// TwinCAT 3 PLC project TcoKukaRobotics
// Title: TcoKukaRobotics
// Company: Vortex.Library
// Author: TcOpenGroup
// ProjectVersion: 0.6.0.913
// ProgramVersion: 3.1.4024.12
// libraries:
//   Tc2_MC2, * (Beckhoff Automation GmbH)
//   Tc2_MC2_Drive, * (Beckhoff Automation GmbH)
//   Tc2_Standard, * (Beckhoff Automation GmbH)
//   Tc2_System, * (Beckhoff Automation GmbH)
//   Tc3_Module, * (Beckhoff Automation GmbH)
//   TcoAbstractions, 0.6.0.913 (Vortex.Library)
//   TcoCore, 0.6.0.913 (Vortex.Library)
//   TcoIo, 0.6.0.913 (Vortex.Library)
//   TcoUtilities, 0.6.0.913 (Vortex.Library)
// project tree:
//   DUTs/ TcoKukaRobotics_Config_v_5_x_x.TcDUT, TcoKukaRobotics_Control_v_5_x_x.TcDUT, TcoKukaRobotics_State_v_5_x_x.TcDUT, TcoKukaRobotics_Status_v_5_x_x.TcDUT
//   / PlcTask.TcTTO
//   POUs/ MAIN.TcPOU
//   POUs/Prototypes/KRC4/IO/ TcoKrc4_Inputs_v_5_x_x.TcDUT, TcoKrc4_IO_v_5_x_x.TcDUT, TcoKrc4_Outputs_v_5_x_x.TcDUT
//   POUs/Prototypes/KRC4/ TcoKrc4_v_5_x_x.TcPOU
//   POUs/Prototypes/RoboticsTasks/Starts/ StartAtMainTask.TcPOU, StartMotorsAndProgramTask.TcPOU, StartMotorsProgramAndMovementsTask.TcPOU, StartMotorsTask.TcPOU, StartMovementsTask.TcPOU, StartProgramTask.TcPOU
//   POUs/Prototypes/RoboticsTasks/Stops/ StopMotorsTask.TcPOU, StopMovementsAndProgramTask.TcPOU, StopMovementsTask.TcPOU, StopProgramTask.TcPOU
//   POUs/Prototypes/RoboticsTasks/ TcoKukaRoboticsTask.TcPOU
// real-time tasks:
//   TASK PlcTask: cycle T#10ms, priority 20, ADS port 350
//   TASK PlcTask1: cycle T#10ms, priority 1, ADS port 351
//   TASK PN: cycle T#8ms, priority 2, ADS port 301
// I/O:
//   DEVICE Device 4 (EtherCAT) (disabled), AmsNetId 172.20.10.104.5.1
//     Term 1 (EK1100) [EK1100 EtherCAT Coupler (2A E-Bus)]
//       Term 2 (EL1008) [EL1008 8Ch. Dig. Input 24V, 3ms]
//       Term 3 (EL2008) [EL2008 8Ch. Dig. Output 24V, 0.5A]
//       Term 4 (EL3052) [EL3052 2Ch. Ana. Input 4-20mA]
//       Term 5 (EL9576) [EL9576 Brake chopper terminal]
//       Term 6 (EL7211-0010) [EL7211-0010 1Ch. MDP742 Servo motor output stage with OCT (50V, 4.5A RMS)]
//       Term 14 (EL7047) [EL7047 1Ch. Stepper motor output stage (50V, 5A)]
//       Term 8 (EL9011) [EL9011 End Terminal]
//   DEVICE Device 1 (EtherCAT) (disabled), AmsNetId 192.168.4.1.2.1
//     Drive 7 (IndraDrive MPB20) [IndraDrive MPB20]
//   DEVICE Device 2 (EtherCAT) (disabled), AmsNetId 192.168.4.1.3.1
//     Term 1 (EK1200) [EK1200-5000 EtherCAT Power supply (2A E-Bus)]
//       Term 10 (EK1122) [EK1122 2 port EtherCAT junction]
//       Term 13 (EL6631) [EL6631 PROFINET IO Controller]
//       Term 12 (EL1809) [EL1809 16Ch. Dig. Input 24V, 3ms]
//       Term 13 (EL2809) [EL2809 16Ch. Dig. Output 24V, 0.5A]
//       Term 15 (EL4004) [EL4004 4Ch. Ana. Output 0-10V, 12bit]
//       Term 16 (EL7342) [EL7342 2Ch. DC motor output stage (50V, 3.5A)]
//       Term 17 (EL4004) [EL4004 4Ch. Ana. Output 0-10V, 12bit]
//       Term 18 (EL6001) [EL6001 Interface (RS232)]
//       Term 10 (EL9011) [EL9011 End Terminal]
//   DEVICE Device 3 (EL6631) (disabled), AmsNetId 192.168.4.1.4.1
//     krc4 [KUKA Roboter GmbH PROFINET IO 0x300]
//       modules: Term 4 (DAP Module), Term 5 (64 safe digital in- and outputs), Term 6 (512 digital in- and outputs)
// variable links:
//   TcoKukaRoboticsTests/TcoKukaRoboticsTests Instance <-> Device 3 (EL6631)/krc4
//     PlcTask1 Inputs/GVL.Robot1.In.Inputs[{0..63}] <-> API/Term 6 (512 digital in- and outputs)/Subterm 10 (512 digital in- and outputs)/Inputs/8 digital inputs[{0..63}]  (64 links)
//     PlcTask1 Inputs/GVL.Robot1.PnIoBoxDiag <-> Inputs/PnIoBoxDiag
//     PlcTask1 Inputs/GVL.Robot1.PnIoBoxState <-> Inputs/PnIoBoxState
//     PlcTask1 Outputs/GVL.Robot1.Out.Outputs[{0..63}] <-> API/Term 6 (512 digital in- and outputs)/Subterm 10 (512 digital in- and outputs)/Outputs/8 digital outputs[{0..63}]  (64 links)

CONFIGURATION TcoKukaRobotics
    RESOURCE PLC ON TwinCAT3
        TASK PlcTask(INTERVAL := T#10ms, PRIORITY := 20);
        PROGRAM MAIN WITH PlcTask : MAIN;
    END_RESOURCE
END_CONFIGURATION

// ---- DUTs/TcoKukaRobotics_Config_v_5_x_x.TcDUT
TYPE TcoKukaRobotics_Config_v_5_x_x :
STRUCT
    InfoTime : TIME := T#2S;
    ErrorTime : TIME := T#0S;
END_STRUCT
END_TYPE

// ---- DUTs/TcoKukaRobotics_Control_v_5_x_x.TcDUT
TYPE TcoKukaRobotics_Control_v_5_x_x :
STRUCT
    {attribute addProperty Name "<#Program Start [EXT_START]#>"}
    ExternalStart : BOOL;
    {attribute addProperty Name "<#Move Enable [MOVE_ENABLE]#>"}
    MoveEnable : BOOL;
    {attribute addProperty Name "<#Error Confirmation [CONF_MESS]#>"}
    ErrorConfirmation : BOOL;
    {attribute addProperty Name "<#Drives Off [DRIVES_OFF]#>"}
    DrivesOff : BOOL;
    {attribute addProperty Name "<#Drives On [DRIVES_ON]#>"}
    DrivesOn : BOOL;
    {attribute addProperty Name "<#Activate Interface [I_O_ACT]#>"}
    ActivateInterface : BOOL;
    {attribute addProperty Name "<#Start At Main [START_AT_MAIN]#>"}
    StartAtMain : BOOL;
    {attribute addProperty Name "<#Master mode#>"}
    MasterMode : BYTE;
    {attribute addProperty Name "<#Tool 1 retract#>"}
    Tool_1_Retract : BOOL;
    {attribute addProperty Name "<#Tool 1 extend#>"}
    Tool_1_Extend : BOOL;
    {attribute addProperty Name "<#Tool 2 retract#>"}
    Tool_2_Retract : BOOL;
    {attribute addProperty Name "<#Tool 2 extend#>"}
    Tool_2_Extend : BOOL;
    {attribute addProperty Name "<#Tool 3 retract#>"}
    Tool_3_Retract : BOOL;
    {attribute addProperty Name "<#Tool 3 extend#>"}
    Tool_3_Extend : BOOL;
    {attribute addProperty Name "<#Tool 4 retract#>"}
    Tool_4_Retract : BOOL;
    {attribute addProperty Name "<#Tool 4 extend#>"}
    Tool_4_Extend : BOOL;
    {attribute addProperty Name "<#Zones#>"}
    Zone : BYTE;
    {attribute addProperty Name "<#In position#>"}
    InPosition : BYTE;
    {attribute addProperty Name "<#Action number#>"}
    ActionNo : BYTE;
    {attribute addProperty Name "<#Global robot speed#>"}
    GlobalSpeed : BYTE;
    {attribute addProperty Name "<#Tool number#>"}
    ToolNo : BYTE;
    {attribute addProperty Name "<#Workobject number#>"}
    WorkobjectNo : BYTE;
    {attribute addProperty Name "<#Point number#>"}
    PointNo : BYTE;
    {attribute addProperty Name "<#User specific speed 1#>"}
    UserSpecSpeed1 : REAL;
    {attribute addProperty Name "<#User specific speed 2#>"}
    UserSpecSpeed2 : REAL;
    {attribute  addProperty Name "<#Coordinates#>"}
    Coordinates : TcoAbstractions.TcoRoboticsCoordinates;
END_STRUCT
END_TYPE

// ---- DUTs/TcoKukaRobotics_State_v_5_x_x.TcDUT
TYPE TcoKukaRobotics_State_v_5_x_x :
STRUCT
    {attribute addProperty Name "<#ControlReady [RC_RDY1]#>"}
    RcReady : BOOL;
    {attribute addProperty Name "<#AlarmStopActive [ALARM_STOP]#>"}
    AlarmStopActive : BOOL;
    {attribute addProperty Name "<#UserSafetySwitchClosed [USER_SAF]#>"}
    UserSafetySwitchClosed : BOOL;
    {attribute addProperty Name "<#DrivesReady [PERI_RDY]#>"}
    DrivesReady : BOOL;
    {attribute addProperty Name "<#RobotCalibrated [ROB_CAL]#>"}
    RobotCalibrated : BOOL;
    {attribute addProperty Name "<#InterfaceActivated [I_O_ACTCONF]#>"}
    InterfaceActivated : BOOL;
    {attribute addProperty Name "<#ErrorCollection [STOPMESS]#>"}
    StopMess : BOOL;
    {attribute addProperty Name "<#RobotStopped [ROB_STOPPED]#>"}
    RobotStopped : BOOL;
    {attribute addProperty Name "<#InHome [IN_HOME]#>"}
    InHome : BOOL;
    {attribute addProperty Name "<#Manual [T1]#>"}
    Manual : BOOL;
    {attribute addProperty Name "<#Automatic [AUT]#>"}
    Automatic : BOOL;
    {attribute addProperty Name "<#ExternalAutomatic [EXT]#>"}
    ExternalAutomatic : BOOL;
    {attribute addProperty Name "<#ProcesActive [PRO_ACT]#>"}
    ProActive : BOOL;
    {attribute addProperty Name "<#ProgramMoveActive [PROGRAM MOVEMENT ACTIVE]#>"}
    ProgramMoveActive : BOOL;
    {attribute addProperty Name "<#Event ID#>"}
    EventId : UDINT;
    {attribute addProperty Name "<#PpMoved#>"}
    PpMoved : BOOL;
    {attribute addProperty Name "<#StartAtMain#>"}
    StartAtMain : BOOL;
    {attribute addProperty Name "<#Error#>"}
    Error : BOOL;
    {attribute addProperty Name "<#In area 1#>"}
    InArea_1 : BOOL;
    {attribute addProperty Name "<#In area 2#>"}
    InArea_2 : BOOL;
    {attribute addProperty Name "<#In area 3#>"}
    InArea_3 : BOOL;
    {attribute addProperty Name "<#In area 4#>"}
    InArea_4 : BOOL;
    {attribute addProperty Name "<#In position 1#>"}
    InPosition_1 : BOOL;
    {attribute addProperty Name "<#In position 2#>"}
    InPosition_2 : BOOL;
    {attribute addProperty Name "<#In position 3#>"}
    InPosition_3 : BOOL;
    {attribute addProperty Name "<#In position 4#>"}
    InPosition_4 : BOOL;
    {attribute addProperty Name "<#Zones#>"}
    Zone : BYTE;
    {attribute addProperty Name "<#In position#>"}
    InPosition : BYTE;
    {attribute addProperty Name "<#Tool 1 retract#>"}
    Tool_1_Retract : BOOL;
    {attribute addProperty Name "<#Tool 1 extend#>"}
    Tool_1_Extend : BOOL;
    {attribute addProperty Name "<#Tool 2 retract#>"}
    Tool_2_Retract : BOOL;
    {attribute addProperty Name "<#Tool 2 extend#>"}
    Tool_2_Extend : BOOL;
    {attribute addProperty Name "<#Tool 3 retract#>"}
    Tool_3_Retract : BOOL;
    {attribute addProperty Name "<#Tool 3 extend#>"}
    Tool_3_Extend : BOOL;
    {attribute addProperty Name "<#Tool 4 retract#>"}
    Tool_4_Retract : BOOL;
    {attribute addProperty Name "<#Tool 4 extend#>"}
    Tool_4_Extend : BOOL;
    {attribute addProperty Name "<#Action number#>"}
    ActionNo : BYTE;
    {attribute addProperty Name "<#Global speed#>"}
    GlobalSpeed : BYTE;
    {attribute addProperty Name "<#Tool number#>"}
    ToolNo : BYTE;
    {attribute addProperty Name "<#Workobject number#>"}
    WorkobjectNo : BYTE;
    {attribute addProperty Name "<#PointNumber#>"}
    PointNo : BYTE;
    {attribute addProperty Name "<#User specific speed 1#>"}
    UserSpecSpeed1 : DINT;
    {attribute addProperty Name "<#User specific speed 2#>"}
    UserSpecSpeed2 : DINT;
    {attribute  addProperty Name "<#Coordinates#>"}
    Coordinates : TcoAbstractions.TcoRoboticsCoordinates;
END_STRUCT
END_TYPE

// ---- DUTs/TcoKukaRobotics_Status_v_5_x_x.TcDUT
TYPE TcoKukaRobotics_Status_v_5_x_x :
STRUCT
    ActionDescription : STRING(100);
    State : TcoKukaRobotics_State_v_5_x_x;
END_STRUCT
END_TYPE

// ---- POUs/Prototypes/KRC4/IO/TcoKrc4_Inputs_v_5_x_x.TcDUT
TYPE TcoKrc4_Inputs_v_5_x_x :
STRUCT
    Inputs AT %I* : ARRAY[0..63] OF BYTE;
END_STRUCT
END_TYPE

// ---- POUs/Prototypes/KRC4/IO/TcoKrc4_IO_v_5_x_x.TcDUT
TYPE TcoKrc4_IO_v_5_x_x :
STRUCT
    PnIoBoxState AT %I* : UINT;
    PnIoBoxDiag AT %I* : UINT;
    PnIoBoxCtrl AT %Q* : UINT;
    {attribute addProperty Name "<#IN#>"}
    In : TcoKrc4_Inputs_v_5_x_x;
    {attribute addProperty Name "<#OUT#>"}
    Out : TcoKrc4_Outputs_v_5_x_x;
END_STRUCT
END_TYPE

// ---- POUs/Prototypes/KRC4/IO/TcoKrc4_Outputs_v_5_x_x.TcDUT
TYPE TcoKrc4_Outputs_v_5_x_x :
STRUCT
    Outputs AT %Q* : ARRAY[0..63] OF BYTE;
END_STRUCT
END_TYPE

// ---- POUs/MAIN.TcPOU
PROGRAM MAIN
VAR
END_VAR

END_PROGRAM

// ---- POUs/Prototypes/KRC4/TcoKrc4_v_5_x_x.TcPOU
FUNCTION_BLOCK TcoKrc4_v_5_x_x EXTENDS TcoIo.TcoPnIoComponent IMPLEMENTS TcoAbstractions.ITcoRobotics
VAR_INPUT
    inEnable : BOOL;
END_VAR
VAR_OUTPUT
END_VAR
VAR_IN_OUT
    inoData : TcoKrc4_IO_v_5_x_x;
END_VAR
VAR
    {attribute addProperty Name "<#Status#>"}
    {attribute clr [ReadOnly()]}
    _status : TcoKukaRobotics_Status_v_5_x_x;
    {attribute addProperty Name "<#Control#>"}
    _control : TcoKukaRobotics_Control_v_5_x_x;
    {attribute addProperty Name "<#Config#>"}
    _config : TcoKukaRobotics_Config_v_5_x_x;
    {attribute addProperty Name "<#PN Error#>"}
    {attribute clr [ReadOnly()]}
    _pnError : BOOL;
    _someTaskIsActive : BOOL;
    _stopTasksAreActive : BOOL;
END_VAR
VAR
    {attribute addProperty Name "<#Start at Main#>"}
    _startAtMainTask : StartAtMainTask(THIS^);
    {attribute addProperty Name "<#Start motors and program#>"}
    _startMotorsAndProgramTask : StartMotorsAndProgramTask(THIS^);
    {attribute addProperty Name "<#Start program#>"}
    _startProgramTask : StartProgramTask(THIS^);
    {attribute addProperty Name "<#Start motors#>"}
    _startMotorsTask : StartMotorsTask(THIS^);
    {attribute addProperty Name "<#Start movements#>"}
    _startMovementsTask : StartMovementsTask(THIS^);
    {attribute addProperty Name "<#Start motors program and movements#>"}
    _startMotorsProgramAndMovementsTask : StartMotorsProgramAndMovementsTask(THIS^);
    {attribute addProperty Name "<#Stop movements#>"}
    _stopMovementsTask : StopMovementsTask(THIS^);
    {attribute addProperty Name "<#Stop movenents and program#>"}
    _stopMovementsAndProgramTask : StopMovementsAndProgramTask(THIS^);
    {attribute addProperty Name "<#Stop program#>"}
    _stopProgramTask : StopProgramTask(THIS^);
    {attribute addProperty Name "<#Stop motors#>"}
    _stopMotorsTask : StopMotorsTask(THIS^);
    {attribute addProperty Name "<#Restore#>"}
    _restoreTask : TcoCore.TcoTask(THIS^);
END_VAR
VAR
    {attribute 'hide'}
    _sb : TcoCore.StringBuilder;
END_VAR

IF NOT __ISVALIDREF(inoData) THEN
    Messenger.Post('Invalid reference', TcoCore.eMessageCategory.ProgrammingError);
    RETURN;
END_IF

SUPER^(inPnIoBoxState := THIS^.inoData.PnIoBoxState, inPnIoBoxDiag := THIS^.inoData.PnIoBoxDiag);
_pnError := not _profinetReady;
UpdateStatus();
_stopTasksAreActive := _stopMovementsTask.Busy AND _stopMovementsAndProgramTask.Busy AND _stopProgramTask.Busy AND _stopMotorsTask.Busy;
_startAtMainTask.Enabled := NOT _stopTasksAreActive;
_startAtMainTask(inoConfig := _config, inoControl := _control, inoStatus := _status);
_startProgramTask.Enabled := NOT _stopTasksAreActive;
_startProgramTask(inoConfig := _config, inoControl := _control, inoStatus := _status);
_startMotorsTask.Enabled := NOT _stopTasksAreActive AND NOT _startMotorsProgramAndMovementsTask.Busy AND NOT _startMotorsAndProgramTask.Busy;
_startMotorsTask(inoConfig := _config, inoControl := _control, inoStatus := _status);
_startMotorsAndProgramTask.Enabled := NOT _stopTasksAreActive AND NOT _startProgramTask.Busy AND NOT _startMotorsTask.Busy;
_startMotorsAndProgramTask(inoConfig := _config, inoControl := _control, inoStatus := _status);
_startMovementsTask.Enabled := NOT _startMotorsProgramAndMovementsTask.Busy AND NOT _stopMotorsTask.Busy;
_startMovementsTask(inoConfig := _config, inoControl := _control, inoStatus := _status);
_startMotorsProgramAndMovementsTask.Enabled := NOT _startMovementsTask.Busy AND NOT _stopMotorsTask.Busy;

_startMotorsProgramAndMovementsTask(refStartMotorsAndProgramTask := _startMotorsAndProgramTask,
    inoConfig := _config,
    inoControl := _control,
    inoStatus := _status);

_stopMovementsTask.Enabled := TRUE;
_stopMovementsTask(inoConfig := _config, inoControl := _control, inoStatus := _status);
_stopMotorsTask.Enabled := TRUE;
_stopMotorsTask(inoConfig := _config, inoControl := _control, inoStatus := _status);
_stopProgramTask.Enabled := TRUE;
_stopProgramTask(inoConfig := _config, inoControl := _control, inoStatus := _status);
_stopMovementsAndProgramTask.Enabled := NOT _stopProgramTask.Busy AND NOT _stopProgramTask.Busy;
_stopMovementsAndProgramTask(inoConfig := _config, inoControl := _control, inoStatus := _status);
//*************RESTORE********************
_restoreTask.Enabled := TRUE;

IF _restoreTask.Execute() THEN
    Restore();
    _restoreTask.DoneWhen(TRUE);
END_IF

//****************************************
_someTaskIsActive := _startAtMainTask.Busy OR
    _startMotorsAndProgramTask.Busy OR
    _startMovementsTask.Busy OR
    _startMovementsTask.Busy OR
    _stopMovementsTask.Busy OR
    _stopMovementsAndProgramTask.Busy OR
    _stopProgramTask.Busy;

//do not publish diagnostic message when component is not used
IF _someTaskIsActive THEN
    IF (NOT _status.State.AlarmStopActive) THEN
        Messenger.Error('<#Emergency stop active#>');
    END_IF;

    IF (NOT _status.State.UserSafetySwitchClosed) THEN
        Messenger.Warning('<#Safety Error #>');
    END_IF;
END_IF;

IF (_status.State.Error) THEN
    Messenger.Error(_sb.Clear()
            .Append('<#Robot reported an error: #>')
            .Append(UDINT_TO_STRING(_status.State.EventId))
            .Append(' |[[0]AdvancedDiagnosticMessage]|')
            .Append('.')
            .Append('For details see the service mode')
            .ToString());
END_IF;

UpdateControl();

(*~
    <docu>
        <summary>
            Gets the configuration of the IRC 5.
        </summary>
    </docu>
~*)
PROPERTY Config : REFERENCE TO TcoKukaRobotics_Config_v_5_x_x
GET
Config REF= _config;
END_GET
END_PROPERTY

PROPERTY PUBLIC Control : REFERENCE TO TcoKukaRobotics_Control_v_5_x_x
GET
Control REF= _control;
END_GET
END_PROPERTY

METHOD FB_init : BOOL
VAR_INPUT
    bInitRetains : BOOL; // if TRUE, the retain variables are initialized (warm start / cold start)
    bInCopyCode : BOOL; // if TRUE, the instance afterwards gets moved into the copy code (online change)
    ParentObject : ITcoObject;
END_VAR
END_METHOD

(*~
    <docu>
        <summary>
            Restores this instance to the Ready state. Can be called explicitly or from within one of the restore mechanisms.
        </summary>
    </docu>
~*)
METHOD Restore : ITcoRestorable
RestoreTasks();
_control.GlobalSpeed := 0;
_control.ActivateInterface := FALSE;
_control.ErrorConfirmation := FALSE;
_control.ExternalStart := FALSE;
_control.MasterMode := 0;
//todo to restore control signals
_control.ToolNo := 0;
_control.WorkobjectNo := 0;
_control.PointNo := 0;
_control.UserSpecSpeed1 := 0;
_control.UserSpecSpeed2 := 0;
_control.Coordinates.X := 0;
_control.Coordinates.Y := 0;
_control.Coordinates.Z := 0;
_control.Coordinates.Rx := 0;
_control.Coordinates.Ry := 0;
_control.Coordinates.Rz := 0;
END_METHOD

METHOD INTERNAL RestoreTasks
//_resetTask.Restore();
_startAtMainTask.Restore();
_startMovementsTask.Restore();
_startProgramTask.Restore();
_startMotorsTask.Restore();
_stopMotorsTask.Restore();
_startMotorsProgramAndMovementsTask.Restore();
_stopMovementsTask.Restore();
_startMotorsAndProgramTask.Restore();
_stopMovementsAndProgramTask.Restore();
_stopProgramTask.Restore();
END_METHOD

(*~
    <docu>
        <summary>
            Custom service (manual, maintenance) logic.
            This method must be implemented in derived class.
        </summary>
    </docu>
~*)
METHOD PROTECTED ServiceMode
END_METHOD

METHOD PUBLIC StartAtMain : TcoCore.ITcoTaskStatus
VAR_INPUT
END_VAR
StartAtMain := _startAtMainTask.Invoke();
END_METHOD

PROPERTY StartAtMainTask : TcoCore.ITcoTaskStatus
GET
StartAtMainTask := _startAtMainTask;
END_GET
END_PROPERTY

METHOD PUBLIC StartMotors : TcoCore.ITcoTaskStatus
StartMotors := _startMotorsTask.Invoke();
END_METHOD

METHOD StartMotorsAndProgram : TcoCore.ITcoTaskStatus
VAR_INPUT
END_VAR
StartMotorsAndProgram := THIS^._startMotorsAndProgramTask.Invoke();
END_METHOD

PROPERTY StartMotorsAndProgramTask : TcoCore.ITcoTaskStatus
GET
StartMotorsAndProgramTask := _startMotorsAndProgramTask;
END_GET
END_PROPERTY

METHOD PUBLIC StartMotorsProgramAndMovements : TcoCore.ITcoTaskStatus
VAR_INPUT
    inData : TcoRoboticsMovementsParams;
END_VAR
StartMotorsProgramAndMovements := _startMotorsProgramAndMovementsTask.InvokeWithParams(inData);
END_METHOD

PROPERTY StartMotorsProgramAndMovementsTask : TcoCore.ITcoTaskStatus
GET
StartMotorsProgramAndMovementsTask := _startMotorsProgramAndMovementsTask;
END_GET
END_PROPERTY

PROPERTY StartMotorsTask : TcoCore.ITcoTaskStatus
GET
StartMotorsTask := _startMotorsTask;
END_GET
END_PROPERTY

METHOD PUBLIC StartMovements : TcoCore.ITcoTaskStatus
VAR_INPUT
    inData : TcoRoboticsMovementsParams;
END_VAR
StartMovements := _startMovementsTask.InvokeWithParams(inData);
END_METHOD

PROPERTY StartMovementsTask : TcoCore.ITcoTaskStatus
GET
StartMovementsTask := _startMovementsTask;
END_GET
END_PROPERTY

METHOD PUBLIC StartProgram : TcoCore.ITcoTaskStatus
StartProgram := _startProgramTask.Invoke();
END_METHOD

PROPERTY StartProgramTask : TcoCore.ITcoTaskStatus
GET
StartProgramTask := _startProgramTask;
END_GET
END_PROPERTY

(*~
    <docu>
        <summary>
            Gets the status of the IRC5.
        </summary>
    </docu>
~*)
PROPERTY Status : REFERENCE TO TcoKukaRobotics_Status_v_5_x_x
GET
Status REF= _status;
END_GET
END_PROPERTY

METHOD PUBLIC StopMotors : TcoCore.ITcoTaskStatus
StopMotors := _stopMotorsTask.Invoke();
END_METHOD

PROPERTY StopMotorsTask : TcoCore.ITcoTaskStatus
GET
StopMotorsTask := _stopMotorsTask;
END_GET
END_PROPERTY

METHOD PUBLIC StopMovements : TcoCore.ITcoTaskStatus
VAR_INPUT
    inStopType : eTcoRoboticsStopType;
END_VAR
StopMovements := _stopMovementsTask.InvokeWithParams(inStopType);
END_METHOD

METHOD PUBLIC StopMovementsAndProgram : TcoCore.ITcoTaskStatus
VAR_INPUT
    inStopType : eTcoRoboticsStopType;
END_VAR
StopMovementsAndProgram := _stopMovementsAndProgramTask.InvokeWithParams(inStopType);
END_METHOD

PROPERTY StopMovementsAndProgramTask : TcoCore.ITcoTaskStatus
GET
StopMovementsAndProgramTask := _stopMovementsAndProgramTask;
END_GET
END_PROPERTY

PROPERTY StopMovementsTask : TcoCore.ITcoTaskStatus
GET
StopMovementsTask := _stopMovementsTask;
END_GET
END_PROPERTY

METHOD PUBLIC StopProgram : TcoCore.ITcoTaskStatus
StopProgram := _stopProgramTask.Invoke();
END_METHOD

PROPERTY StopProgramTask : TcoCore.ITcoTaskStatus
GET
StopProgramTask := _stopProgramTask;
END_GET
END_PROPERTY

METHOD INTERNAL UpdateControl
VAR_INPUT
END_VAR
VAR
    index : INT;
END_VAR
//SYSTEM OUTPUTS
index := 0;
inoData.Out.Outputs[index].0 := _control.ExternalStart;
inoData.Out.Outputs[index].1 := _control.MoveEnable;
inoData.Out.Outputs[index].2 := _control.ErrorConfirmation;
inoData.Out.Outputs[index].3 := _control.DrivesOff;
inoData.Out.Outputs[index].4 := _control.DrivesOn;
inoData.Out.Outputs[index].5 := _control.ActivateInterface;
inoData.Out.Outputs[index].6 := _control.StartAtMain;
//index:=1;
//inoData.Out.Outputs[index].0 	:= 		_control.StartProgram;
//inoData.Out.Outputs[index].1 	:= 		_control.StartAtMain;
//inoData.Out.Outputs[index].2 	:= 		_control.StopProgram;
//inoData.Out.Outputs[index].3 	:= 		_control.QuickStop;
//inoData.Out.Outputs[index].4 	:= 		_control.SoftStop;
//inoData.Out.Outputs[index].5 	:= 		_control.StopCycle;
//inoData.Out.Outputs[index].6 	:= 		_control.StopInstruction;
//inoData.Out.Outputs[index].7 	:= 		_control.LimitSpeed;
//Tool signals
index := 2;
inoData.Out.Outputs[index].0 := _control.Tool_1_Retract;
inoData.Out.Outputs[index].1 := _control.Tool_1_Extend;
inoData.Out.Outputs[index].2 := _control.Tool_2_Retract;
inoData.Out.Outputs[index].3 := _control.Tool_2_Extend;
inoData.Out.Outputs[index].4 := _control.Tool_3_Retract;
inoData.Out.Outputs[index].5 := _control.Tool_3_Extend;
inoData.Out.Outputs[index].6 := _control.Tool_4_Retract;
inoData.Out.Outputs[index].7 := _control.Tool_4_Extend;
//master mode  such as manual/auto ....
index := 3;
inoData.Out.Outputs[index] := _control.MasterMode;
//zone
index := 5;
inoData.Out.Outputs[index] := _control.Zone;
//position
index := 6;
inoData.Out.Outputs[index] := _control.InPosition;
//
//Movement parameters
index := 7;
inoData.Out.Outputs[index] := _control.ActionNo;
index := 8;
inoData.Out.Outputs[index] := _control.GlobalSpeed;
index := 9;
inoData.Out.Outputs[index] := _control.ToolNo;
index := 10;
inoData.Out.Outputs[index] := _control.WorkobjectNo;
index := 11;
inoData.Out.Outputs[index] := _control.PointNo;
index := 12;

TcoUtilities.TcoDintToBytes(inFormat := TcoUtilities.eTcoDataFormat.LittleEndian,
    inValue := REAL_TO_DINT(_control.UserSpecSpeed1),
    outByte0 := inoData.Out.Outputs[index],
    outByte1 := inoData.Out.Outputs[index + 1],
    outByte2 := inoData.Out.Outputs[index + 2],
    outByte3 := inoData.Out.Outputs[index + 3]);

index := 16;

TcoUtilities.TcoDintToBytes(inFormat := TcoUtilities.eTcoDataFormat.LittleEndian,
    inValue := REAL_TO_DINT(_control.UserSpecSpeed2),
    outByte0 := inoData.Out.Outputs[index],
    outByte1 := inoData.Out.Outputs[index + 1],
    outByte2 := inoData.Out.Outputs[index + 2],
    outByte3 := inoData.Out.Outputs[index + 3]);
////Coordinates
index := 20;

TcoUtilities.TcoDintToBytes(inFormat := TcoUtilities.eTcoDataFormat.LittleEndian,
    inValue := REAL_TO_DINT((_control.Coordinates.X) * 10000.0),
    outByte0 := inoData.Out.Outputs[index],
    outByte1 := inoData.Out.Outputs[index + 1],
    outByte2 := inoData.Out.Outputs[index + 2],
    outByte3 := inoData.Out.Outputs[index + 3]);

index := 24;

TcoUtilities.TcoDintToBytes(inFormat := TcoUtilities.eTcoDataFormat.LittleEndian,
    inValue := REAL_TO_DINT((_control.Coordinates.Y) * 10000.0),
    outByte0 := inoData.Out.Outputs[index],
    outByte1 := inoData.Out.Outputs[index + 1],
    outByte2 := inoData.Out.Outputs[index + 2],
    outByte3 := inoData.Out.Outputs[index + 3]);

index := 28;

TcoUtilities.TcoDintToBytes(inFormat := TcoUtilities.eTcoDataFormat.LittleEndian,
    inValue := REAL_TO_DINT((_control.Coordinates.Z) * 10000.0),
    outByte0 := inoData.Out.Outputs[index],
    outByte1 := inoData.Out.Outputs[index + 1],
    outByte2 := inoData.Out.Outputs[index + 2],
    outByte3 := inoData.Out.Outputs[index + 3]);

index := 32;

TcoUtilities.TcoDintToBytes(inFormat := TcoUtilities.eTcoDataFormat.LittleEndian,
    inValue := REAL_TO_DINT((_control.Coordinates.Rx) * 10000.0),
    outByte0 := inoData.Out.Outputs[index],
    outByte1 := inoData.Out.Outputs[index + 1],
    outByte2 := inoData.Out.Outputs[index + 2],
    outByte3 := inoData.Out.Outputs[index + 3]);

index := 36;

TcoUtilities.TcoDintToBytes(inFormat := TcoUtilities.eTcoDataFormat.LittleEndian,
    inValue := REAL_TO_DINT((_control.Coordinates.Ry) * 10000.0),
    outByte0 := inoData.Out.Outputs[index],
    outByte1 := inoData.Out.Outputs[index + 1],
    outByte2 := inoData.Out.Outputs[index + 2],
    outByte3 := inoData.Out.Outputs[index + 3]);

index := 40;

TcoUtilities.TcoDintToBytes(inFormat := TcoUtilities.eTcoDataFormat.LittleEndian,
    inValue := REAL_TO_DINT((_control.Coordinates.Rz) * 10000.0),
    outByte0 := inoData.Out.Outputs[index],
    outByte1 := inoData.Out.Outputs[index + 1],
    outByte2 := inoData.Out.Outputs[index + 2],
    outByte3 := inoData.Out.Outputs[index + 3]);
END_METHOD

METHOD INTERNAL UpdateStatus
VAR
    _message : STRING(125);
    tempOut : BYTE;
    index : INT;
    _bytes : DINT;
END_VAR
//SYSTEM INPUTS
index := 0;
_status.State.RcReady := inoData.In.Inputs[index].0;
_status.State.AlarmStopActive := inoData.In.Inputs[index].1;
_status.State.UserSafetySwitchClosed := inoData.In.Inputs[index].2;
_status.State.DrivesReady := inoData.In.Inputs[index].3;
_status.State.RobotCalibrated := inoData.In.Inputs[index].4;
_status.State.InterfaceActivated := inoData.In.Inputs[index].5;
_status.State.StopMess := inoData.In.Inputs[index].6;
_status.State.RobotStopped := inoData.In.Inputs[index].7;
index := 1;
_status.State.InHome := inoData.In.Inputs[index].0;
_status.State.Manual := inoData.In.Inputs[index].1;
_status.State.Automatic := inoData.In.Inputs[index].2;
_status.State.ExternalAutomatic := inoData.In.Inputs[index].3;
_status.State.ProActive := inoData.In.Inputs[index].4;
_status.State.PpMoved := inoData.In.Inputs[index].5;
_status.State.Error := inoData.In.Inputs[index].6;
_status.State.ProgramMoveActive := inoData.In.Inputs[index].7;
//Area/positions flags this  should be obsolete because Zones and InPosition is used as byte below
index := 2;
_status.State.InArea_1 := inoData.In.Inputs[index].0;
_status.State.InArea_2 := inoData.In.Inputs[index].1;
_status.State.InArea_3 := inoData.In.Inputs[index].2;
_status.State.InArea_4 := inoData.In.Inputs[index].3;
_status.State.InPosition_1 := inoData.In.Inputs[index].4;
_status.State.InPosition_2 := inoData.In.Inputs[index].5;
_status.State.InPosition_3 := inoData.In.Inputs[index].6;
_status.State.InPosition_4 := inoData.In.Inputs[index].7;
//
//Tool signals
index := 3;
_status.State.Tool_1_Retract := inoData.In.Inputs[index].0;
_status.State.Tool_1_Extend := inoData.In.Inputs[index].1;
_status.State.Tool_2_Retract := inoData.In.Inputs[index].2;
_status.State.Tool_2_Extend := inoData.In.Inputs[index].3;
_status.State.Tool_3_Retract := inoData.In.Inputs[index].4;
_status.State.Tool_3_Extend := inoData.In.Inputs[index].5;
_status.State.Tool_4_Retract := inoData.In.Inputs[index].6;
_status.State.Tool_4_Extend := inoData.In.Inputs[index].7;
//Safety signals
index := 4;
index := 5;
_status.State.Zone := inoData.In.Inputs[index];
index := 6;
_status.State.InPosition := inoData.In.Inputs[index];
//Movement parameters
index := 7;
_status.State.ActionNo := inoData.In.Inputs[index];
index := 8;
_status.State.GlobalSpeed := inoData.In.Inputs[index];
index := 9;
_status.State.ToolNo := inoData.In.Inputs[index];
index := 10;
_status.State.WorkobjectNo := inoData.In.Inputs[index];
index := 11;
_status.State.PointNo := inoData.In.Inputs[index];
index := 12;

_status.State.UserSpecSpeed1 := TcoUtilities.TcoBytesToDint(inFormat := TcoUtilities.eTcoDataFormat.LittleEndian,
    inByte0 := inoData.In.Inputs[index],
    inByte1 := inoData.In.Inputs[index + 1],
    inByte2 := inoData.In.Inputs[index + 2],
    inByte3 := inoData.In.Inputs[index + 3]);

index := 16;

_status.State.UserSpecSpeed2 := TcoUtilities.TcoBytesToDint(inFormat := TcoUtilities.eTcoDataFormat.LittleEndian,
    inByte0 := inoData.In.Inputs[index],
    inByte1 := inoData.In.Inputs[index + 1],
    inByte2 := inoData.In.Inputs[index + 2],
    inByte3 := inoData.In.Inputs[index + 3]);

index := 20;

_bytes := TcoUtilities.TcoBytesToDint(inFormat := TcoUtilities.eTcoDataFormat.LittleEndian,
    inByte0 := inoData.In.Inputs[index],
    inByte1 := inoData.In.Inputs[index + 1],
    inByte2 := inoData.In.Inputs[index + 2],
    inByte3 := inoData.In.Inputs[index + 3]);

_status.State.Coordinates.X := (DINT_TO_REAL(_bytes) / 10000.0);
index := 24;

_bytes := TcoUtilities.TcoBytesToDint(inFormat := TcoUtilities.eTcoDataFormat.LittleEndian,
    inByte0 := inoData.In.Inputs[index],
    inByte1 := inoData.In.Inputs[index + 1],
    inByte2 := inoData.In.Inputs[index + 2],
    inByte3 := inoData.In.Inputs[index + 3]);

_status.State.Coordinates.Y := (DINT_TO_REAL(_bytes) / 10000.0);
index := 28;

_bytes := TcoUtilities.TcoBytesToDint(inFormat := TcoUtilities.eTcoDataFormat.LittleEndian,
    inByte0 := inoData.In.Inputs[index],
    inByte1 := inoData.In.Inputs[index + 1],
    inByte2 := inoData.In.Inputs[index + 2],
    inByte3 := inoData.In.Inputs[index + 3]);

_status.State.Coordinates.Z := (DINT_TO_REAL(_bytes) / 10000.0);
index := 32;

_bytes := TcoUtilities.TcoBytesToDint(inFormat := TcoUtilities.eTcoDataFormat.LittleEndian,
    inByte0 := inoData.In.Inputs[index],
    inByte1 := inoData.In.Inputs[index + 1],
    inByte2 := inoData.In.Inputs[index + 2],
    inByte3 := inoData.In.Inputs[index + 3]);

_status.State.Coordinates.Rx := (DINT_TO_REAL(_bytes) / 10000.0);
index := 36;

_bytes := TcoUtilities.TcoBytesToDint(inFormat := TcoUtilities.eTcoDataFormat.LittleEndian,
    inByte0 := inoData.In.Inputs[index],
    inByte1 := inoData.In.Inputs[index + 1],
    inByte2 := inoData.In.Inputs[index + 2],
    inByte3 := inoData.In.Inputs[index + 3]);

_status.State.Coordinates.Ry := (DINT_TO_REAL(_bytes) / 10000.0);
index := 40;

_bytes := TcoUtilities.TcoBytesToDint(inFormat := TcoUtilities.eTcoDataFormat.LittleEndian,
    inByte0 := inoData.In.Inputs[index],
    inByte1 := inoData.In.Inputs[index + 1],
    inByte2 := inoData.In.Inputs[index + 2],
    inByte3 := inoData.In.Inputs[index + 3]);

_status.State.Coordinates.Rz := (DINT_TO_REAL(_bytes) / 10000.0);
index := 44;

_status.State.EventId := TcoUtilities.TcoBytesToUDint(inFormat := TcoUtilities.eTcoDataFormat.LittleEndian,
    inByte0 := inoData.In.Inputs[index],
    inByte1 := inoData.In.Inputs[index + 1],
    inByte2 := inoData.In.Inputs[index + 2],
    inByte3 := inoData.In.Inputs[index + 3]);
END_METHOD

END_FUNCTION_BLOCK

// ---- POUs/Prototypes/RoboticsTasks/Starts/StartAtMainTask.TcPOU
FUNCTION_BLOCK StartAtMainTask EXTENDS TcoKukaRoboticsTask

IF Execute() THEN
    _blink(inOnTime := T#500MS, inOffTime := T#500MS);

    IF _progress = 0 THEN
        IF NOT __ISVALIDREF(inoControl) THEN
            _varInfo := __VARINFO(inoControl);
            Messenger.Programming(_sb.Clear().Append('<#Invalid reference: #>').Append(_varInfo.Symbol).ToString()).Pin();
        ELSIF NOT __ISVALIDREF(inoConfig) THEN
            _varInfo := __VARINFO(inoConfig);
            Messenger.Programming(_sb.Clear().Append('<#Invalid reference: #>').Append(_varInfo.Symbol).ToString()).Pin();
        ELSIF NOT __ISVALIDREF(inoStatus) THEN
            _varInfo := __VARINFO(inoStatus);
            Messenger.Programming(_sb.Clear().Append('<#Invalid reference: #>').Append(_varInfo.Symbol).ToString()).Pin();
        ELSE
            _progress := _progress + 1;
        END_IF
    END_IF

    IF _progress = 1 THEN
        inoControl.StartAtMain := not inoStatus.State.PpMoved and _blink.outQ;
        _varInfo := __VARINFO(inoStatus.State.PpMoved);

        THIS^.Messenger.OnCondition(_infoTimer.Q AND NOT inoStatus.State.PpMoved)
            .Warning(_sb.Clear().Append('<#Waiting program pointer changed! #>').Append(_varInfo.Symbol).ToString());

        IF inoStatus.State.PpMoved THEN
            inoControl.StartAtMain := FALSE;
            _progress := 0;
        END_IF
    END_IF

    DoneWhen(inoStatus.State.PpMoved);
    CallTimers(TRUE);
    THIS^.ThrowWhen(_errorTimer.Q);
END_IF;

IF THIS^.Error AND NOT _errorMessage.Pinned THEN
    THIS^.Restore();
END_IF

METHOD PUBLIC FB_init : BOOL
VAR_INPUT
    bInitRetains : BOOL; // if TRUE, the retain variables are initialized (warm start / cold start)
    bInCopyCode : BOOL; // if TRUE, the instance afterwards gets moved into the copy code (online change)
    ParentObject : ITcoObject;
END_VAR
END_METHOD

(*~
    <docu>
        <summary>
            Executes when task is aborted.
        </summary>
    </docu>
~*)
METHOD PROTECTED OnAbort
IF __ISVALIDREF(inoStatus) THEN
    THIS^.inoStatus.ActionDescription := '<#Start at Main was aborted, while not yet completed!#>';
END_IF;
END_METHOD

(*~
    <docu>
        <summary>
            Executes when task reaches the ```Done``` state .
        </summary>
    </docu>
~*)
METHOD PROTECTED OnDone
IF __ISVALIDREF(inoStatus) THEN
    THIS^.inoStatus.ActionDescription := '<#Start at Main was completed successfully.#>';
END_IF;
END_METHOD

(*~
    <docu>
        <summary>
            Executes when task reaches the ```Error``` state.
            <para>
                Do not confuse with <see cref="PlcDocu.TcoCore.TcoTask.WhileError()"/>, that is called cyclically until '''Error''' state is left.
            </para>
        </summary>
    </docu>
~*)
METHOD PROTECTED OnError
VAR
    description : STRING;
END_VAR
description := '<#Start at Main finished with error.#>';

IF __ISVALIDREF(inoStatus) THEN
    THIS^.inoStatus.ActionDescription := description;
END_IF;

THIS^._errorMessage.Error(_sb.Clear().Append(description).Append(' To restore acknowledge this alarm.').ToString()).Pin();
END_METHOD

METHOD PROTECTED OnStart
IF __ISVALIDREF(inoStatus) THEN
    THIS^.inoStatus.ActionDescription := '<#Start at Main started.#>';
END_IF;

inoControl.ActionNo := 255;
END_METHOD

(*~
    <docu>
        <summary>
            Restores this instance to the Ready state. Can be called explicitly or from within one of the restore mechanisms.
            <para>
                See also <see cref="PlcDocu.TcoCore.TcoTask.AutoRestorable()"/>
            </para>
        </summary>
    </docu>
~*)
METHOD Restore : ITcoRestorable
SUPER^.Restore();
END_METHOD

END_FUNCTION_BLOCK

// ---- POUs/Prototypes/RoboticsTasks/TcoKukaRoboticsTask.TcPOU
FUNCTION_BLOCK PUBLIC ABSTRACT TcoKukaRoboticsTask EXTENDS TcoCore.TcoTask
VAR_IN_OUT
    inoConfig : TcoKukaRobotics_Config_v_5_x_x;
    inoControl : TcoKukaRobotics_Control_v_5_x_x;
    inoStatus : TcoKukaRobotics_Status_v_5_x_x;
END_VAR
VAR
    _errorMessage : TcoCore.TcoMessenger(THIS^);
    {attribute 'hide'}
    _progress : INT := 0;
    {attribute 'hide'}
    _infoTimer : TON;
    {attribute 'hide'}
    _errorTimer : TON;
    {attribute 'hide'}
    _timer : TON;
    {attribute 'hide'}
    _varInfo : __SYSTEM.VAR_INFO;
    {attribute 'hide'}
    _sb : TcoCore.StringBuilder;
    {attribute 'hide'}
    _blink : TcoUtilities.TcoBlinker(THIS^);
END_VAR

METHOD CallTimers
VAR_INPUT
    inValue : BOOL;
END_VAR
IF __ISVALIDREF(inoConfig) AND THIS^.inoConfig.ErrorTime <> T#0S OR NOT inValue THEN
    _errorTimer(IN := inValue, PT := THIS^.inoConfig.ErrorTime);
END_IF;

IF __ISVALIDREF(inoConfig) AND THIS^.inoConfig.InfoTime <> T#0S OR NOT inValue THEN
    _infoTimer(IN := inValue, PT := THIS^.inoConfig.InfoTime);
END_IF;
END_METHOD

(*~
    <docu>
        <summary>
            Restores this instance to the Ready state. Can be called explicitly or from within one of the restore mechanisms.
            <para>
                See also <see cref="PlcDocu.TcoCore.TcoTask.AutoRestorable()"/>
            </para>
        </summary>
    </docu>
~*)
METHOD Restore : ITcoRestorable
SUPER^.Restore();
_progress := 0;
_timer(In := FALSE);
CallTimers(FALSE);
Messenger.UnPin();
_errorMessage.UnPin();
END_METHOD

END_FUNCTION_BLOCK

// ---- POUs/Prototypes/RoboticsTasks/Starts/StartMotorsAndProgramTask.TcPOU
FUNCTION_BLOCK StartMotorsAndProgramTask EXTENDS TcoKukaRoboticsTask

IF Execute() THEN
    _blink(inOnTime := T#500MS, inOffTime := T#500MS);

    IF _progress = 0 THEN
        IF NOT __ISVALIDREF(inoControl) THEN
            _varInfo := __VARINFO(inoControl);
            Messenger.Programming(_sb.Clear().Append('<#Invalid reference: #>').Append(_varInfo.Symbol).ToString()).Pin();
        ELSIF NOT __ISVALIDREF(inoConfig) THEN
            _varInfo := __VARINFO(inoConfig);
            Messenger.Programming(_sb.Clear().Append('<#Invalid reference: #>').Append(_varInfo.Symbol).ToString()).Pin();
        ELSIF NOT __ISVALIDREF(inoStatus) THEN
            _varInfo := __VARINFO(inoStatus);
            Messenger.Programming(_sb.Clear().Append('<#Invalid reference: #>').Append(_varInfo.Symbol).ToString()).Pin();
        ELSE
            _progress := _progress + 1;
        END_IF
    END_IF

    IF _progress = 1 THEN
        _varInfo := __VARINFO(inoStatus.State.UserSafetySwitchClosed);

        THIS^.Messenger.OnCondition(_infoTimer.Q AND NOT inoStatus.State.UserSafetySwitchClosed)
            .Warning(_sb.Clear().Append('<#Waiting for signal#>').Append(_varInfo.Symbol).ToString());

        IF inoStatus.State.UserSafetySwitchClosed THEN
            _progress := _progress + 1;
        END_IF;
    END_IF;

    IF _progress = 2 THEN
        _varInfo := __VARINFO(inoStatus.State.AlarmStopActive);

        THIS^.Messenger.OnCondition(_infoTimer.Q AND NOT inoStatus.State.AlarmStopActive)
            .Warning(_sb.Clear().Append('<#Waiting for signal#>').Append(_varInfo.Symbol).ToString());

        IF inoStatus.State.AlarmStopActive THEN
            _progress := _progress + 1;
        END_IF;
    END_IF;

    IF _progress = 3 THEN
        _varInfo := __VARINFO(inoStatus.State.DrivesReady);

        THIS^.Messenger.OnCondition(_infoTimer.Q AND NOT inoStatus.State.DrivesReady)
            .Warning(_sb.Clear().Append('<# Waiting for signal: #>').Append(_varInfo.Symbol).ToString());

        inoControl.DrivesOff := TRUE;
        inoControl.DrivesOn := _blink.outQ;

        IF inoStatus.State.DrivesReady THEN
            inoControl.DrivesOn := FALSE;
            _progress := _progress + 1;
        END_IF
    END_IF;

    IF _progress = 4 THEN
        Messenger.Debug('<#Robot Error Reset and Move Enable#>');
        inoControl.MoveEnable := TRUE;
        inoControl.ErrorConfirmation := inoStatus.State.StopMess AND _blink.outQ;
        _varInfo := __VARINFO(inoStatus.State.StopMess);

        THIS^.Messenger.OnCondition(_infoTimer.Q AND inoStatus.State.StopMess)
            .Warning(_sb.Clear().Append('<#Waiting for signal#>').Append(_varInfo.Symbol).Append(' is OFF').ToString());

        _varInfo := __VARINFO(inoStatus.State.RcReady);

        THIS^.Messenger.OnCondition(_infoTimer.Q AND NOT inoStatus.State.RcReady)
            .Warning(_sb.Clear().Append('<#Waiting for signal#>').Append(_varInfo.Symbol).ToString());

        IF NOT inoStatus.State.StopMess AND inoStatus.State.RcReady THEN
            inoControl.ErrorConfirmation := FALSE;
            _progress := _progress + 1;
        END_IF
    END_IF;

    IF _progress = 5 THEN
        inoControl.ActivateInterface := TRUE;
        _varInfo := __VARINFO(inoStatus.State.InterfaceActivated);

        THIS^.Messenger.OnCondition(_infoTimer.Q AND NOT inoStatus.State.InterfaceActivated)
            .Warning(_sb.Clear().Append('<#Waiting for signal#>').Append(_varInfo.Symbol).ToString());

        IF inoStatus.State.InterfaceActivated THEN
            _progress := _progress + 1;
        END_IF;
    END_IF;

    IF _progress = 6 THEN
        IF inoStatus.State.StopMess OR inoStatus.State.AlarmStopActive OR NOT inoStatus.State.RcReady THEN
            _progress := 1;
        END_IF

        inoControl.ExternalStart := _blink.outQ;
        _varInfo := __VARINFO(inoStatus.State.ProActive);

        THIS^.Messenger.OnCondition(_infoTimer.Q AND NOT inoStatus.State.ProActive)
            .Warning(_sb.Clear().Append('<#Waiting for program running signal! #>').Append(_varInfo.Symbol).ToString());

        IF inoStatus.State.ProActive THEN
            inoControl.ExternalStart := FALSE;
        END_IF
    END_IF;

    DoneWhen(inoStatus.State.ProActive AND inoStatus.State.DrivesReady AND NOT inoStatus.State.StopMess);
    CallTimers(TRUE);
    THIS^.ThrowWhen(_errorTimer.Q);
END_IF

IF THIS^.Error AND NOT _errorMessage.Pinned THEN
    THIS^.Restore();
END_IF

METHOD PUBLIC FB_init : BOOL
VAR_INPUT
    bInitRetains : BOOL; // if TRUE, the retain variables are initialized (warm start / cold start)
    bInCopyCode : BOOL; // if TRUE, the instance afterwards gets moved into the copy code (online change)
    ParentObject : ITcoObject;
END_VAR
END_METHOD

(*~
    <docu>
        <summary>
            Executes when task is aborted.
        </summary>
    </docu>
~*)
METHOD PROTECTED OnAbort
IF __ISVALIDREF(inoStatus) THEN
    THIS^.inoStatus.ActionDescription := '<#Start motors and program was aborted.#>';
END_IF;
END_METHOD

(*~
    <docu>
        <summary>
            Executes when task reaches the ```Done``` state .
        </summary>
    </docu>
~*)
METHOD PROTECTED OnDone
IF __ISVALIDREF(inoStatus) THEN
    THIS^.inoStatus.ActionDescription := '<#Start motors and program finished successfully.#>';
END_IF;

_progress := 0;
inoControl.ActivateInterface := FALSE;
END_METHOD

METHOD PROTECTED OnError
VAR
    description : STRING;
END_VAR
description := '<#Start motors and program finished with error.#>';

IF __ISVALIDREF(inoStatus) THEN
    THIS^.inoStatus.ActionDescription := description;
END_IF;

THIS^._errorMessage.Error(_sb.Clear().Append(description).Append(' To restore acknowledge this alarm.').ToString()).Pin();
END_METHOD

METHOD PROTECTED OnStart
IF __ISVALIDREF(inoStatus) THEN
    THIS^.inoStatus.ActionDescription := '<#Start motors and program started.#>';
END_IF;

CallTimers(FALSE);
inoControl.MoveEnable := TRUE;
END_METHOD

(*~
    <docu>
        <summary>
            Restores this instance to the Ready state. Can be called explicitly or from within one of the restore mechanisms.
            <para>
                See also <see cref="PlcDocu.TcoCore.TcoTask.AutoRestorable()"/>
            </para>
        </summary>
    </docu>
~*)
METHOD Restore : ITcoRestorable
SUPER^.Restore();
END_METHOD

END_FUNCTION_BLOCK

// ---- POUs/Prototypes/RoboticsTasks/Starts/StartProgramTask.TcPOU
FUNCTION_BLOCK StartProgramTask EXTENDS TcoKukaRoboticsTask
VAR
    _stopType : TcoAbstractions.eTcoRoboticsStopType;
END_VAR

IF Execute() THEN
    _blink(inOnTime := T#500MS, inOffTime := T#500MS);

    IF _progress = 0 THEN
        IF NOT __ISVALIDREF(inoControl) THEN
            _varInfo := __VARINFO(inoControl);
            Messenger.Programming(_sb.Clear().Append('<#Invalid reference: #>').Append(_varInfo.Symbol).ToString()).Pin();
        ELSIF NOT __ISVALIDREF(inoConfig) THEN
            _varInfo := __VARINFO(inoConfig);
            Messenger.Programming(_sb.Clear().Append('<#Invalid reference: #>').Append(_varInfo.Symbol).ToString()).Pin();
        ELSIF NOT __ISVALIDREF(inoStatus) THEN
            _varInfo := __VARINFO(inoStatus);
            Messenger.Programming(_sb.Clear().Append('<#Invalid reference: #>').Append(_varInfo.Symbol).ToString()).Pin();
        ELSE
            _progress := _progress + 1;
        END_IF
    END_IF

    IF _progress = 1 THEN
        _varInfo := __VARINFO(inoStatus.State.UserSafetySwitchClosed);

        THIS^.Messenger.OnCondition(_infoTimer.Q AND NOT inoStatus.State.UserSafetySwitchClosed)
            .Warning(_sb.Clear().Append('<#Waiting for signal#>').Append(_varInfo.Symbol).ToString());

        IF inoStatus.State.UserSafetySwitchClosed THEN
            _progress := _progress + 1;
        END_IF;
    END_IF;

    IF _progress = 2 THEN
        _varInfo := __VARINFO(inoStatus.State.AlarmStopActive);

        THIS^.Messenger.OnCondition(_infoTimer.Q AND NOT inoStatus.State.AlarmStopActive)
            .Warning(_sb.Clear().Append('<#Waiting for signal#>').Append(_varInfo.Symbol).ToString());

        IF inoStatus.State.AlarmStopActive THEN
            _progress := _progress + 1;
        END_IF;
    END_IF;

    IF _progress = 3 THEN
        _varInfo := __VARINFO(inoStatus.State.DrivesReady);

        THIS^.Messenger.OnCondition(_infoTimer.Q AND NOT inoStatus.State.DrivesReady)
            .Warning(_sb.Clear().Append('<# Waiting for signal: #>').Append(_varInfo.Symbol).ToString());

        inoControl.DrivesOff := TRUE;
        inoControl.DrivesOn := _blink.outQ;

        IF inoStatus.State.DrivesReady THEN
            inoControl.DrivesOn := FALSE;
            _progress := _progress + 1;
        END_IF
    END_IF;

    IF _progress = 4 THEN
        Messenger.Debug('<#Robot Error Reset and Move Enable#>');
        inoControl.MoveEnable := TRUE;
        inoControl.ErrorConfirmation := inoStatus.State.StopMess AND _blink.outQ;
        _varInfo := __VARINFO(inoStatus.State.StopMess);

        THIS^.Messenger.OnCondition(_infoTimer.Q AND inoStatus.State.StopMess)
            .Warning(_sb.Clear().Append('<#Waiting for signal#>').Append(_varInfo.Symbol).Append(' is OFF').ToString());

        _varInfo := __VARINFO(inoStatus.State.RcReady);

        THIS^.Messenger.OnCondition(_infoTimer.Q AND NOT inoStatus.State.RcReady)
            .Warning(_sb.Clear().Append('<#Waiting for signal#>').Append(_varInfo.Symbol).ToString());

        IF NOT inoStatus.State.StopMess AND inoStatus.State.RcReady THEN
            inoControl.ErrorConfirmation := FALSE;
            _progress := _progress + 1;
        END_IF
    END_IF;

    IF _progress = 5 THEN
        inoControl.ActivateInterface := TRUE;
        _varInfo := __VARINFO(inoStatus.State.InterfaceActivated);

        THIS^.Messenger.OnCondition(_infoTimer.Q AND NOT inoStatus.State.InterfaceActivated)
            .Warning(_sb.Clear().Append('<#Waiting for signal#>').Append(_varInfo.Symbol).ToString());

        IF inoStatus.State.InterfaceActivated THEN
            _progress := _progress + 1;
        END_IF;
    END_IF;

    IF _progress = 6 THEN
        IF inoStatus.State.StopMess OR inoStatus.State.AlarmStopActive OR NOT inoStatus.State.RcReady THEN
            _progress := 1;
        END_IF

        inoControl.ExternalStart := _blink.outQ;
        _varInfo := __VARINFO(inoStatus.State.ProActive);

        THIS^.Messenger.OnCondition(_infoTimer.Q AND NOT inoStatus.State.ProActive)
            .Warning(_sb.Clear().Append('<#Waiting for program running signal! #>').Append(_varInfo.Symbol).ToString());

        IF inoStatus.State.ProActive THEN
            inoControl.ExternalStart := FALSE;
        END_IF
    END_IF;

    DoneWhen(inoStatus.State.ProActive AND inoStatus.State.DrivesReady AND NOT inoStatus.State.StopMess);
    CallTimers(TRUE);
    THIS^.ThrowWhen(_errorTimer.Q);
END_IF

IF THIS^.Error AND NOT _errorMessage.Pinned THEN
    THIS^.Restore();
END_IF

METHOD PUBLIC FB_init : BOOL
VAR_INPUT
    bInitRetains : BOOL; // if TRUE, the retain variables are initialized (warm start / cold start)
    bInCopyCode : BOOL; // if TRUE, the instance afterwards gets moved into the copy code (online change)
    ParentObject : ITcoObject;
END_VAR
END_METHOD

METHOD INTERNAL InvokeWithParams : ITcoTaskStatus
VAR_INPUT
    inStopType : eTcoRoboticsStopType;
END_VAR
_stopType := inStopType;
InvokeWithParams := THIS^.Invoke();
END_METHOD

(*~
    <docu>
        <summary>
            Executes when task is aborted.
        </summary>
    </docu>
~*)
METHOD PROTECTED OnAbort
IF __ISVALIDREF(inoStatus) THEN
    THIS^.inoStatus.ActionDescription := '<#Stop program was aborted, while not yet completed!#>';
END_IF;
END_METHOD

(*~
    <docu>
        <summary>
            Executes when task reaches the ```Done``` state .
        </summary>
    </docu>
~*)
METHOD PROTECTED OnDone
IF __ISVALIDREF(inoStatus) THEN
    THIS^.inoStatus.ActionDescription := '<#Stop program was completed successfully.#>';
END_IF;

_progress := 0;
inoControl.ActivateInterface := FALSE;
END_METHOD

(*~
    <docu>
        <summary>
            Executes when task reaches the ```Error``` state.
                </summary>
    </docu>
~*)
METHOD PROTECTED OnError
VAR
    description : STRING;
END_VAR
THIS^.inoStatus.ActionDescription := '<#Stopping program with error.#>';

IF __ISVALIDREF(inoStatus) THEN
    THIS^.inoStatus.ActionDescription := description;
END_IF;

THIS^._errorMessage.Error(_sb.Clear().Append(description).Append(' To restore acknowledge this alarm.').ToString()).Pin();
END_METHOD

METHOD PROTECTED OnStart
IF __ISVALIDREF(inoStatus) THEN
    THIS^.inoStatus.ActionDescription := '<#Stopping program started.#>';
END_IF;

CallTimers(FALSE);
END_METHOD

(*~
    <docu>
        <summary>
            Restores this instance to the Ready state. Can be called explicitly or from within one of the restore mechanisms.
            <para>
                See also <see cref="PlcDocu.TcoCore.TcoTask.AutoRestorable()"/>
            </para>
        </summary>
    </docu>
~*)
METHOD Restore : ITcoRestorable
SUPER^.Restore();
END_METHOD

END_FUNCTION_BLOCK

// ---- POUs/Prototypes/RoboticsTasks/Starts/StartMotorsTask.TcPOU
FUNCTION_BLOCK StartMotorsTask EXTENDS TcoKukaRoboticsTask

IF Execute() THEN
    _blink(inOnTime := T#500MS, inOffTime := T#500MS);

    IF _progress = 0 THEN
        IF NOT __ISVALIDREF(inoControl) THEN
            _varInfo := __VARINFO(inoControl);
            Messenger.Programming(_sb.Clear().Append('<#Invalid reference: #>').Append(_varInfo.Symbol).ToString()).Pin();
        ELSIF NOT __ISVALIDREF(inoConfig) THEN
            _varInfo := __VARINFO(inoConfig);
            Messenger.Programming(_sb.Clear().Append('<#Invalid reference: #>').Append(_varInfo.Symbol).ToString()).Pin();
        ELSIF NOT __ISVALIDREF(inoStatus) THEN
            _varInfo := __VARINFO(inoStatus);
            Messenger.Programming(_sb.Clear().Append('<#Invalid reference: #>').Append(_varInfo.Symbol).ToString()).Pin();
        ELSE
            _progress := _progress + 1;
        END_IF
    END_IF

    //	IF _progress = 1 THEN
    //		inoControl.ActivateInterface:=TRUE;
    //		_varInfo :=__VARINFO( inoStatus.State.InterfaceActivated);
    //		THIS^.Messenger.OnCondition(_infoTimer.Q AND NOT inoStatus.State.InterfaceActivated).Warning(_sb.Clear().Append('<#Waiting for signal#>').Append(_varInfo.Symbol).ToString());
    //		IF  inoStatus.State.InterfaceActivated THEN
    //			_progress := _progress + 1;
    //		END_IF;
    //	END_IF;
    IF _progress = 1 THEN
        _varInfo := __VARINFO(inoStatus.State.UserSafetySwitchClosed);

        THIS^.Messenger.OnCondition(_infoTimer.Q AND NOT inoStatus.State.UserSafetySwitchClosed)
            .Warning(_sb.Clear().Append('<#Waiting for signal#>').Append(_varInfo.Symbol).ToString());

        IF inoStatus.State.UserSafetySwitchClosed THEN
            _progress := _progress + 1;
        END_IF;
    END_IF;

    IF _progress = 2 THEN
        _varInfo := __VARINFO(inoStatus.State.AlarmStopActive);

        THIS^.Messenger.OnCondition(_infoTimer.Q AND NOT inoStatus.State.AlarmStopActive)
            .Warning(_sb.Clear().Append('<#Waiting for signal#>').Append(_varInfo.Symbol).ToString());

        IF inoStatus.State.AlarmStopActive THEN
            _progress := _progress + 1;
        END_IF;
    END_IF;

    IF _progress = 3 THEN
        _varInfo := __VARINFO(inoStatus.State.DrivesReady);

        THIS^.Messenger.OnCondition(_infoTimer.Q AND NOT inoStatus.State.DrivesReady)
            .Warning(_sb.Clear().Append('<# Waiting for signal: #>').Append(_varInfo.Symbol).ToString());

        inoControl.DrivesOff := TRUE;
        inoControl.DrivesOn := _blink.outQ;

        IF inoStatus.State.DrivesReady THEN
            inoControl.DrivesOn := FALSE;
            _progress := _progress + 1;
        END_IF
    END_IF;

    DoneWhen(inoStatus.State.DrivesReady);
    CallTimers(TRUE);
    THIS^.ThrowWhen(_errorTimer.Q);
END_IF

IF THIS^.Error AND NOT _errorMessage.Pinned THEN
    THIS^.Restore();
END_IF

METHOD PUBLIC FB_init : BOOL
VAR_INPUT
    bInitRetains : BOOL; // if TRUE, the retain variables are initialized (warm start / cold start)
    bInCopyCode : BOOL; // if TRUE, the instance afterwards gets moved into the copy code (online change)
    ParentObject : ITcoObject;
END_VAR
END_METHOD

(*~
    <docu>
        <summary>
            Executes when task is aborted.
        </summary>
    </docu>
~*)
METHOD PROTECTED OnAbort
IF __ISVALIDREF(inoStatus) THEN
    THIS^.inoStatus.ActionDescription := '<#Start motors  was aborted.#>';
END_IF;
END_METHOD

(*~
    <docu>
        <summary>
            Executes when task reaches the ```Done``` state .
        </summary>
    </docu>
~*)
METHOD PROTECTED OnDone
IF __ISVALIDREF(inoStatus) THEN
    THIS^.inoStatus.ActionDescription := '<#Start motors  finished successfully.#>';
END_IF;

_progress := 0;
END_METHOD

METHOD PROTECTED OnError
VAR
    description : STRING;
END_VAR
description := '<#Start motors finished with error.#>';

IF __ISVALIDREF(inoStatus) THEN
    THIS^.inoStatus.ActionDescription := description;
END_IF;

THIS^._errorMessage.Error(_sb.Clear().Append(description).Append(' To restore acknowledge this alarm.').ToString()).Pin();
END_METHOD

METHOD PROTECTED OnStart
IF __ISVALIDREF(inoStatus) THEN
    THIS^.inoStatus.ActionDescription := '<#Start motors started.#>';
END_IF;

CallTimers(FALSE);
END_METHOD

(*~
    <docu>
        <summary>
            Restores this instance to the Ready state. Can be called explicitly or from within one of the restore mechanisms.
            <para>
                See also <see cref="PlcDocu.TcoCore.TcoTask.AutoRestorable()"/>
            </para>
        </summary>
    </docu>
~*)
METHOD Restore : ITcoRestorable
SUPER^.Restore();
END_METHOD

END_FUNCTION_BLOCK

// ---- POUs/Prototypes/RoboticsTasks/Starts/StartMovementsTask.TcPOU
FUNCTION_BLOCK StartMovementsTask EXTENDS TcoKukaRoboticsTask
VAR
    _moveParams : TcoAbstractions.TcoRoboticsMovementsParams;
END_VAR

IF Execute() THEN
    IF _progress = 0 THEN
        IF NOT __ISVALIDREF(inoControl) THEN
            _varInfo := __VARINFO(inoControl);
            Messenger.Programming(_sb.Clear().Append('<#Invalid reference: #>').Append(_varInfo.Symbol).ToString()).Pin();
        ELSIF NOT __ISVALIDREF(inoConfig) THEN
            _varInfo := __VARINFO(inoConfig);
            Messenger.Programming(_sb.Clear().Append('<#Invalid reference: #>').Append(_varInfo.Symbol).ToString()).Pin();
        ELSIF NOT __ISVALIDREF(inoStatus) THEN
            _varInfo := __VARINFO(inoStatus);
            Messenger.Programming(_sb.Clear().Append('<#Invalid reference: #>').Append(_varInfo.Symbol).ToString()).Pin();
        ELSE
            _progress := _progress + 1;
        END_IF
    END_IF

    IF _progress = 1 THEN
        _varInfo := __VARINFO(inoStatus.State.ProActive);

        THIS^.Messenger.OnCondition(_infoTimer.Q AND NOT inoStatus.State.ProActive)
            .Warning(_sb.Clear().Append('<#Waiting for program running signal! #>').Append(_varInfo.Symbol).ToString());

        _varInfo := __VARINFO(inoStatus.State.DrivesReady);

        THIS^.Messenger.OnCondition(_infoTimer.Q AND NOT inoStatus.State.DrivesReady)
            .Warning(_sb.Clear().Append('<#Waiting for motors are On! #>').Append(_varInfo.Symbol).ToString());

        _varInfo := __VARINFO(inoStatus.State.StopMess);

        THIS^.Messenger.OnCondition(_infoTimer.Q AND inoStatus.State.StopMess)
            .Warning(_sb.Clear().Append('<#Waiting for system is without errors! #>').Append(_varInfo.Symbol).ToString());

        IF inoStatus.State.ProActive AND inoStatus.State.DrivesReady AND NOT inoStatus.State.StopMess THEN
            _progress := _progress + 1;
        END_IF
    END_IF;

    IF _progress = 2 THEN
        inoControl.GlobalSpeed := _moveParams.GlobalSpeed;
        inoControl.ToolNo := _moveParams.ToolNo;
        inoControl.WorkobjectNo := _moveParams.WorkobjectNo;
        inoControl.PointNo := _moveParams.PointNo;
        inoControl.UserSpecSpeed1 := _moveParams.UserSpecSpeed1;
        inoControl.UserSpecSpeed2 := _moveParams.UserSpecSpeed2;
        inoControl.Coordinates := _moveParams.Coordinates;
        inoControl.ActionNo := 254;

        IF inoControl.ActionNo = inoStatus.State.ActionNo THEN
            _progress := _progress + 1;
        END_IF
    END_IF;

    IF _progress = 3 THEN
        IF inoStatus.State.GlobalSpeed = _moveParams.GlobalSpeed AND
            inoStatus.State.ToolNo = _moveParams.ToolNo AND
            inoStatus.State.WorkobjectNo = _moveParams.WorkobjectNo AND
            inoStatus.State.PointNo = _moveParams.PointNo AND
            inoStatus.State.UserSpecSpeed1 = _moveParams.UserSpecSpeed1 AND
            inoStatus.State.UserSpecSpeed2 = _moveParams.UserSpecSpeed2 AND
            TcoAbstractions.CoordinatesAreEqual(inoStatus.State.Coordinates,
                _moveParams.Coordinates,
                0.01,
                0.01,
                0.01,
                0.01,
                0.01,
                0.01) THEN
            inoControl.ActionNo := 253;
            _progress := _progress + 1;
        END_IF
    END_IF;

    IF _progress = 4 THEN
        IF inoControl.ActionNo = inoStatus.State.ActionNo THEN
            _progress := _progress + 1;
        END_IF
    END_IF;

    IF _progress = 5 THEN
        Messenger.Info(CONCAT('<#Moving to position ID#>: ', INT_TO_STRING(_moveParams.ActionNo)));
        inoControl.ActionNo := _moveParams.ActionNo;

        IF inoControl.ActionNo = inoStatus.State.ActionNo THEN
            inoControl.ActionNo := 255;
            _progress := _progress + 1;
        END_IF
    END_IF;

    IF _progress = 6 THEN
        IF inoControl.ActionNo = inoStatus.State.ActionNo THEN
            DoneWhen(TRUE);
        END_IF
    END_IF;

    CallTimers(TRUE);
    THIS^.ThrowWhen(_errorTimer.Q);
END_IF

IF THIS^.Error AND NOT _errorMessage.Pinned THEN
    THIS^.Restore();
END_IF

METHOD PUBLIC FB_init : BOOL
VAR_INPUT
    bInitRetains : BOOL; // if TRUE, the retain variables are initialized (warm start / cold start)
    bInCopyCode : BOOL; // if TRUE, the instance afterwards gets moved into the copy code (online change)
    ParentObject : ITcoObject;
END_VAR
END_METHOD

METHOD INTERNAL InvokeWithParams : ITcoTaskStatus
VAR_INPUT
    inMoveParams : TcoAbstractions.TcoRoboticsMovementsParams;
END_VAR
_moveParams := inMoveParams;
InvokeWithParams := THIS^.Invoke();
END_METHOD

(*~
    <docu>
        <summary>
            Executes when task is aborted.
        </summary>
    </docu>
~*)
METHOD PROTECTED OnAbort
IF __ISVALIDREF(inoStatus) THEN
    THIS^.inoStatus.ActionDescription := '<#Start movements was aborted, while not yet completed!#>';
END_IF;

inoControl.MoveEnable := FALSE;
END_METHOD

(*~
    <docu>
        <summary>
            Executes when task reaches the ```Done``` state .
        </summary>
    </docu>
~*)
METHOD PROTECTED OnDone
IF __ISVALIDREF(inoStatus) THEN
    THIS^.inoStatus.ActionDescription := '<#Start movements finished successfully.#>';
END_IF;

_progress := 0;
END_METHOD

(*~
    <docu>
        <summary>
            Executes when task reaches the ```Error``` state.

        </summary>
    </docu>
~*)
METHOD PROTECTED OnError
VAR
    description : STRING;
END_VAR
description := '<#Start movements finished with error.#>';

IF __ISVALIDREF(inoStatus) THEN
    THIS^.inoStatus.ActionDescription := description;
END_IF;

THIS^._errorMessage.Error(_sb.Clear().Append(description).Append(' To restore acknowledge this alarm.').ToString()).Pin();
END_METHOD

METHOD PROTECTED OnStart
IF __ISVALIDREF(inoStatus) THEN
    THIS^.inoStatus.ActionDescription := '<#Start movements stared.#>';
END_IF;

CallTimers(FALSE);
END_METHOD

(*~
    <docu>
        <summary>
            Restores this instance to the Ready state. Can be called explicitly or from within one of the restore mechanisms.
            <para>
                See also <see cref="PlcDocu.TcoCore.TcoTask.AutoRestorable()"/>
            </para>
        </summary>
    </docu>
~*)
METHOD Restore : ITcoRestorable
SUPER^.Restore();
END_METHOD

END_FUNCTION_BLOCK

// ---- POUs/Prototypes/RoboticsTasks/Starts/StartMotorsProgramAndMovementsTask.TcPOU
FUNCTION_BLOCK StartMotorsProgramAndMovementsTask EXTENDS TcoKukaRoboticsTask
VAR_INPUT
    refStartMotorsAndProgramTask : REFERENCE TO StartMotorsAndProgramTask;
END_VAR
VAR
    _moveParams : TcoAbstractions.TcoRoboticsMovementsParams;
END_VAR
VAR
    _startMotorsAndProgramTask : REFERENCE TO StartMotorsAndProgramTask;
END_VAR

IF NOT __ISVALIDREF(refStartMotorsAndProgramTask) THEN
    Messenger.Post('<#Invalid reference StartMotorAndProgramTask#>', TcoCore.eMessageCategory.ProgrammingError);
    RETURN;
END_IF

_startMotorsAndProgramTask REF= refStartMotorsAndProgramTask;

IF Execute() THEN
    IF _progress = 0 THEN
        IF NOT __ISVALIDREF(inoControl) THEN
            _varInfo := __VARINFO(inoControl);
            Messenger.Programming(_sb.Clear().Append('<#Invalid reference: #>').Append(_varInfo.Symbol).ToString()).Pin();
        ELSIF NOT __ISVALIDREF(inoConfig) THEN
            _varInfo := __VARINFO(inoConfig);
            Messenger.Programming(_sb.Clear().Append('<#Invalid reference: #>').Append(_varInfo.Symbol).ToString()).Pin();
        ELSIF NOT __ISVALIDREF(inoStatus) THEN
            _varInfo := __VARINFO(inoStatus);
            Messenger.Programming(_sb.Clear().Append('<#Invalid reference: #>').Append(_varInfo.Symbol).ToString()).Pin();
        ELSE
            _progress := _progress + 1;
        END_IF
    END_IF

    IF _progress = 1 THEN
        IF _startMotorsAndProgramTask.Invoke().Done THEN
            _progress := _progress + 1;
        END_IF
    END_IF;

    IF _progress = 2 THEN
        inoControl.GlobalSpeed := _moveParams.GlobalSpeed;
        inoControl.ToolNo := _moveParams.ToolNo;
        inoControl.WorkobjectNo := _moveParams.WorkobjectNo;
        inoControl.PointNo := _moveParams.PointNo;
        inoControl.UserSpecSpeed1 := _moveParams.UserSpecSpeed1;
        inoControl.UserSpecSpeed2 := _moveParams.UserSpecSpeed2;
        inoControl.Coordinates := _moveParams.Coordinates;
        inoControl.ActionNo := 254;

        IF inoControl.ActionNo = inoStatus.State.ActionNo THEN
            _progress := _progress + 1;
        END_IF
    END_IF;

    IF _progress = 3 THEN
        IF inoStatus.State.GlobalSpeed = _moveParams.GlobalSpeed AND
            inoStatus.State.ToolNo = _moveParams.ToolNo AND
            inoStatus.State.WorkobjectNo = _moveParams.WorkobjectNo AND
            inoStatus.State.PointNo = _moveParams.PointNo AND
            inoStatus.State.UserSpecSpeed1 = _moveParams.UserSpecSpeed1 AND
            inoStatus.State.UserSpecSpeed2 = _moveParams.UserSpecSpeed2 AND
            TcoAbstractions.CoordinatesAreEqual(inoStatus.State.Coordinates,
                _moveParams.Coordinates,
                0.01,
                0.01,
                0.01,
                0.01,
                0.01,
                0.01) THEN
            inoControl.ActionNo := 253;
            _progress := _progress + 1;
        END_IF
    END_IF;

    IF _progress = 4 THEN
        IF inoControl.ActionNo = inoStatus.State.ActionNo THEN
            _progress := _progress + 1;
        END_IF
    END_IF;

    IF _progress = 5 THEN
        Messenger.Info(CONCAT('<#Moving to position ID#>: ', INT_TO_STRING(_moveParams.ActionNo)));
        inoControl.ActionNo := _moveParams.ActionNo;

        IF inoControl.ActionNo = inoStatus.State.ActionNo THEN
            inoControl.ActionNo := 255;
            _progress := _progress + 1;
        END_IF
    END_IF;

    IF _progress = 6 THEN
        IF inoControl.ActionNo = inoStatus.State.ActionNo THEN
            DoneWhen(TRUE);
        END_IF
    END_IF;

    CallTimers(TRUE);
    THIS^.ThrowWhen(_errorTimer.Q);
END_IF

IF THIS^.Error AND NOT _errorMessage.Pinned THEN
    THIS^.Restore();
END_IF

METHOD PUBLIC FB_init : BOOL
VAR_INPUT
    bInitRetains : BOOL; // if TRUE, the retain variables are initialized (warm start / cold start)
    bInCopyCode : BOOL; // if TRUE, the instance afterwards gets moved into the copy code (online change)
    ParentObject : ITcoObject;
END_VAR
END_METHOD

METHOD INTERNAL InvokeWithParams : ITcoTaskStatus
VAR_INPUT
    inMoveParams : TcoAbstractions.TcoRoboticsMovementsParams;
END_VAR
_moveParams := inMoveParams;
InvokeWithParams := THIS^.Invoke();
END_METHOD

(*~
    <docu>
        <summary>
            Executes when task is aborted.
        </summary>
    </docu>
~*)
METHOD PROTECTED OnAbort
IF __ISVALIDREF(inoStatus) THEN
    THIS^.inoStatus.ActionDescription := '<#Start motors, program and movements was aborted, while not yet completed!#>';
END_IF;
END_METHOD

(*~
    <docu>
        <summary>
            Executes when task reaches the ```Done``` state .
        </summary>
    </docu>
~*)
METHOD PROTECTED OnDone
IF __ISVALIDREF(inoStatus) THEN
    THIS^.inoStatus.ActionDescription := '<#Start motors, program and movements finished successfully.#>';
END_IF;

_progress := 0;
END_METHOD

(*~
    <docu>
        <summary>
            Executes when task reaches the ```Error``` state.
        </summary>
    </docu>
~*)
METHOD PROTECTED OnError
VAR
    description : STRING;
END_VAR
description := '<#Start motors, program and movements finished with error.#>';

IF __ISVALIDREF(inoStatus) THEN
    THIS^.inoStatus.ActionDescription := description;
END_IF;

THIS^._errorMessage.Error(_sb.Clear().Append(description).Append(' To restore acknowledge this alarm.').ToString()).Pin();
END_METHOD

METHOD PROTECTED OnStart
IF __ISVALIDREF(inoStatus) THEN
    THIS^.inoStatus.ActionDescription := '<#Start motors, program and movements stared.#>';
END_IF;

CallTimers(FALSE);
END_METHOD

(*~
    <docu>
        <summary>
            Restores this instance to the Ready state. Can be called explicitly or from within one of the restore mechanisms.
            <para>
                See also <see cref="PlcDocu.TcoCore.TcoTask.AutoRestorable()"/>
            </para>
        </summary>
    </docu>
~*)
METHOD Restore : ITcoRestorable
SUPER^.Restore();
END_METHOD

END_FUNCTION_BLOCK

// ---- POUs/Prototypes/RoboticsTasks/Stops/StopMovementsTask.TcPOU
FUNCTION_BLOCK StopMovementsTask EXTENDS TcoKukaRoboticsTask
VAR
    _stopType : TcoAbstractions.eTcoRoboticsStopType;
END_VAR

IF Execute() THEN
    IF _progress = 0 THEN
        IF NOT __ISVALIDREF(inoControl) THEN
            _varInfo := __VARINFO(inoControl);
            Messenger.Programming(_sb.Clear().Append('<#Invalid reference: #>').Append(_varInfo.Symbol).ToString()).Pin();
        ELSIF NOT __ISVALIDREF(inoConfig) THEN
            _varInfo := __VARINFO(inoConfig);
            Messenger.Programming(_sb.Clear().Append('<#Invalid reference: #>').Append(_varInfo.Symbol).ToString()).Pin();
        ELSIF NOT __ISVALIDREF(inoStatus) THEN
            _varInfo := __VARINFO(inoStatus);
            Messenger.Programming(_sb.Clear().Append('<#Invalid reference: #>').Append(_varInfo.Symbol).ToString()).Pin();
        ELSE
            _progress := _progress + 1;
        END_IF
    END_IF

    IF _progress = 1 THEN
        inoControl.MoveEnable := FALSE;
    END_IF;

    _varInfo := __VARINFO(inoStatus.State.RobotStopped);
    THIS^.Messenger.OnCondition(_infoTimer.Q).Warning(_sb.Clear().Append('<# Waiting for signal: #>').Append(_varInfo.Symbol).ToString());
    DoneWhen(inoStatus.State.RobotStopped);
    CallTimers(TRUE);
    THIS^.ThrowWhen(_errorTimer.Q);
END_IF

IF THIS^.Error AND NOT _errorMessage.Pinned THEN
    THIS^.Restore();
END_IF

METHOD PUBLIC FB_init : BOOL
VAR_INPUT
    bInitRetains : BOOL; // if TRUE, the retain variables are initialized (warm start / cold start)
    bInCopyCode : BOOL; // if TRUE, the instance afterwards gets moved into the copy code (online change)
    ParentObject : ITcoObject;
END_VAR
END_METHOD

METHOD INTERNAL InvokeWithParams : ITcoTaskStatus
VAR_INPUT
    inStopType : eTcoRoboticsStopType;
END_VAR
_stopType := inStopType;
InvokeWithParams := THIS^.Invoke();
END_METHOD

(*~
    <docu>
        <summary>
            Executes when task is aborted.
        </summary>
    </docu>
~*)
METHOD PROTECTED OnAbort
IF __ISVALIDREF(inoStatus) THEN
    THIS^.inoStatus.ActionDescription := '<#Stopping movements was aborted, while not yet completed!#>';
END_IF;

inoControl.MoveEnable := FALSE;
END_METHOD

(*~
    <docu>
        <summary>
            Executes when task reaches the ```Done``` state .
        </summary>
    </docu>
~*)
METHOD PROTECTED OnDone
IF __ISVALIDREF(inoStatus) THEN
    THIS^.inoStatus.ActionDescription := '<#Stopping movements was completed successfully.#>';
END_IF;

_progress := 0;
END_METHOD

(*~
    <docu>
        <summary>
            Executes when task reaches the ```Error``` state.
        </summary>
    </docu>
~*)
METHOD PROTECTED OnError
VAR
    description : STRING;
END_VAR
THIS^.inoStatus.ActionDescription := '<#Stopping movement finished with error.#>';

IF __ISVALIDREF(inoStatus) THEN
    THIS^.inoStatus.ActionDescription := description;
END_IF;

THIS^._errorMessage.Error(_sb.Clear().Append(description).Append(' To restore acknowledge this alarm.').ToString()).Pin();
END_METHOD

METHOD PROTECTED OnStart
IF __ISVALIDREF(inoStatus) THEN
    THIS^.inoStatus.ActionDescription := '<#Stopping movements started.#>';
END_IF;

CallTimers(FALSE);
END_METHOD

(*~
    <docu>
        <summary>
            Restores this instance to the Ready state. Can be called explicitly or from within one of the restore mechanisms.
            <para>
                See also <see cref="PlcDocu.TcoCore.TcoTask.AutoRestorable()"/>
            </para>
        </summary>
    </docu>
~*)
METHOD Restore : ITcoRestorable
SUPER^.Restore();
END_METHOD

END_FUNCTION_BLOCK

// ---- POUs/Prototypes/RoboticsTasks/Stops/StopMovementsAndProgramTask.TcPOU
FUNCTION_BLOCK StopMovementsAndProgramTask EXTENDS TcoKukaRoboticsTask
VAR
    _stopType : TcoAbstractions.eTcoRoboticsStopType;
END_VAR

IF Execute() THEN
    IF _progress = 0 THEN
        IF NOT __ISVALIDREF(inoControl) THEN
            _varInfo := __VARINFO(inoControl);
            Messenger.Programming(_sb.Clear().Append('<#Invalid reference: #>').Append(_varInfo.Symbol).ToString()).Pin();
        ELSIF NOT __ISVALIDREF(inoConfig) THEN
            _varInfo := __VARINFO(inoConfig);
            Messenger.Programming(_sb.Clear().Append('<#Invalid reference: #>').Append(_varInfo.Symbol).ToString()).Pin();
        ELSIF NOT __ISVALIDREF(inoStatus) THEN
            _varInfo := __VARINFO(inoStatus);
            Messenger.Programming(_sb.Clear().Append('<#Invalid reference: #>').Append(_varInfo.Symbol).ToString()).Pin();
        ELSE
            _progress := _progress + 1;
        END_IF
    END_IF

    IF _progress = 1 THEN
        inoControl.MoveEnable := FALSE;
    END_IF;

    _varInfo := __VARINFO(inoStatus.State.RobotStopped);
    THIS^.Messenger.OnCondition(_infoTimer.Q).Warning(_sb.Clear().Append('<# Waiting for signal: #>').Append(_varInfo.Symbol).ToString());
    _varInfo := __VARINFO(inoStatus.State.ProActive);

    THIS^.Messenger.OnCondition(_infoTimer.Q AND inoStatus.State.ProActive)
        .Warning(_sb.Clear().Append('<# Waiting for signal: #>').Append(_varInfo.Symbol).Append('<# is OFF #>').ToString());

    DoneWhen(inoStatus.State.RobotStopped AND NOT inoStatus.State.ProActive);
    CallTimers(TRUE);
    THIS^.ThrowWhen(_errorTimer.Q);
END_IF

IF THIS^.Error AND NOT _errorMessage.Pinned THEN
    THIS^.Restore();
END_IF

METHOD PUBLIC FB_init : BOOL
VAR_INPUT
    bInitRetains : BOOL; // if TRUE, the retain variables are initialized (warm start / cold start)
    bInCopyCode : BOOL; // if TRUE, the instance afterwards gets moved into the copy code (online change)
    ParentObject : ITcoObject;
END_VAR
END_METHOD

METHOD INTERNAL InvokeWithParams : ITcoTaskStatus
VAR_INPUT
    inStopType : eTcoRoboticsStopType;
END_VAR
_stopType := inStopType;
InvokeWithParams := THIS^.Invoke();
END_METHOD

(*~
    <docu>
        <summary>
            Executes when task is aborted.
        </summary>
    </docu>
~*)
METHOD PROTECTED OnAbort
IF __ISVALIDREF(inoStatus) THEN
    THIS^.inoStatus.ActionDescription := '<#Stop movements and program was aborted, while not yet completed!#>';
END_IF;
END_METHOD

(*~
    <docu>
        <summary>
            Executes when task reaches the ```Done``` state .
        </summary>
    </docu>
~*)
METHOD PROTECTED OnDone
IF __ISVALIDREF(inoStatus) THEN
    THIS^.inoStatus.ActionDescription := '<#Stop movements and program  was completed successfully.#>';
END_IF;

_progress := 0;
END_METHOD

(*~
    <docu>
        <summary>
            Executes when task reaches the ```Error``` state.

        </summary>
    </docu>
~*)
METHOD PROTECTED OnError
VAR
    description : STRING;
END_VAR
THIS^.inoStatus.ActionDescription := '<#Stop movements and program finished with error.#>';

IF __ISVALIDREF(inoStatus) THEN
    THIS^.inoStatus.ActionDescription := description;
END_IF;

THIS^._errorMessage.Error(_sb.Clear().Append(description).Append(' To restore acknowledge this alarm.').ToString()).Pin();
END_METHOD

METHOD PROTECTED OnStart
IF __ISVALIDREF(inoStatus) THEN
    THIS^.inoStatus.ActionDescription := '<#Stop movements and program started.#>';
END_IF;

CallTimers(FALSE);
END_METHOD

(*~
    <docu>
        <summary>
            Restores this instance to the Ready state. Can be called explicitly or from within one of the restore mechanisms.
            <para>
                See also <see cref="PlcDocu.TcoCore.TcoTask.AutoRestorable()"/>
            </para>
        </summary>
    </docu>
~*)
METHOD Restore : ITcoRestorable
SUPER^.Restore();
END_METHOD

END_FUNCTION_BLOCK

// ---- POUs/Prototypes/RoboticsTasks/Stops/StopProgramTask.TcPOU
FUNCTION_BLOCK StopProgramTask EXTENDS TcoKukaRoboticsTask
VAR
    _stopType : TcoAbstractions.eTcoRoboticsStopType;
END_VAR

IF Execute() THEN
    IF _progress = 0 THEN
        IF NOT __ISVALIDREF(inoControl) THEN
            _varInfo := __VARINFO(inoControl);
            Messenger.Programming(_sb.Clear().Append('<#Invalid reference: #>').Append(_varInfo.Symbol).ToString()).Pin();
        ELSIF NOT __ISVALIDREF(inoConfig) THEN
            _varInfo := __VARINFO(inoConfig);
            Messenger.Programming(_sb.Clear().Append('<#Invalid reference: #>').Append(_varInfo.Symbol).ToString()).Pin();
        ELSIF NOT __ISVALIDREF(inoStatus) THEN
            _varInfo := __VARINFO(inoStatus);
            Messenger.Programming(_sb.Clear().Append('<#Invalid reference: #>').Append(_varInfo.Symbol).ToString()).Pin();
        ELSE
            _progress := _progress + 1;
        END_IF
    END_IF

    IF _progress = 1 THEN
        inoControl.MoveEnable := FALSE;
    END_IF;

    _varInfo := __VARINFO(inoStatus.State.ProActive);

    THIS^.Messenger.OnCondition(_infoTimer.Q AND inoStatus.State.ProActive)
        .Warning(_sb.Clear().Append('<# Waiting for signal: #>').Append(_varInfo.Symbol).Append('<# is OFF #>').ToString());

    DoneWhen(NOT inoStatus.State.ProActive);
    CallTimers(TRUE);
    THIS^.ThrowWhen(_errorTimer.Q);
END_IF

IF THIS^.Error AND NOT _errorMessage.Pinned THEN
    THIS^.Restore();
END_IF

METHOD PUBLIC FB_init : BOOL
VAR_INPUT
    bInitRetains : BOOL; // if TRUE, the retain variables are initialized (warm start / cold start)
    bInCopyCode : BOOL; // if TRUE, the instance afterwards gets moved into the copy code (online change)
    ParentObject : ITcoObject;
END_VAR
END_METHOD

METHOD INTERNAL InvokeWithParams : ITcoTaskStatus
VAR_INPUT
    inStopType : eTcoRoboticsStopType;
END_VAR
_stopType := inStopType;
InvokeWithParams := THIS^.Invoke();
END_METHOD

(*~
    <docu>
        <summary>
            Executes when task is aborted.
        </summary>
    </docu>
~*)
METHOD PROTECTED OnAbort
IF __ISVALIDREF(inoStatus) THEN
    THIS^.inoStatus.ActionDescription := '<#Stop program was aborted, while not yet completed!#>';
END_IF;
END_METHOD

(*~
    <docu>
        <summary>
            Executes when task reaches the ```Done``` state .
        </summary>
    </docu>
~*)
METHOD PROTECTED OnDone
IF __ISVALIDREF(inoStatus) THEN
    THIS^.inoStatus.ActionDescription := '<#Stop program was completed successfully.#>';
END_IF;

_progress := 0;
END_METHOD

(*~
    <docu>
        <summary>
            Executes when task reaches the ```Error``` state.
>
        </summary>
    </docu>
~*)
METHOD PROTECTED OnError
VAR
    description : STRING;
END_VAR
THIS^.inoStatus.ActionDescription := '<#Stopping program with error.#>';

IF __ISVALIDREF(inoStatus) THEN
    THIS^.inoStatus.ActionDescription := description;
END_IF;

THIS^._errorMessage.Error(_sb.Clear().Append(description).Append(' To restore acknowledge this alarm.').ToString()).Pin();
END_METHOD

METHOD PROTECTED OnStart
IF __ISVALIDREF(inoStatus) THEN
    THIS^.inoStatus.ActionDescription := '<#Stopping program started.#>';
END_IF;

CallTimers(FALSE);
END_METHOD

(*~
    <docu>
        <summary>
            Restores this instance to the Ready state. Can be called explicitly or from within one of the restore mechanisms.
            <para>
                See also <see cref="PlcDocu.TcoCore.TcoTask.AutoRestorable()"/>
            </para>
        </summary>
    </docu>
~*)
METHOD Restore : ITcoRestorable
SUPER^.Restore();
END_METHOD

END_FUNCTION_BLOCK

// ---- POUs/Prototypes/RoboticsTasks/Stops/StopMotorsTask.TcPOU
FUNCTION_BLOCK StopMotorsTask EXTENDS TcoKukaRoboticsTask

IF Execute() THEN
    IF _progress = 0 THEN
        IF NOT __ISVALIDREF(inoControl) THEN
            _varInfo := __VARINFO(inoControl);
            Messenger.Programming(_sb.Clear().Append('<#Invalid reference: #>').Append(_varInfo.Symbol).ToString()).Pin();
        ELSIF NOT __ISVALIDREF(inoConfig) THEN
            _varInfo := __VARINFO(inoConfig);
            Messenger.Programming(_sb.Clear().Append('<#Invalid reference: #>').Append(_varInfo.Symbol).ToString()).Pin();
        ELSIF NOT __ISVALIDREF(inoStatus) THEN
            _varInfo := __VARINFO(inoStatus);
            Messenger.Programming(_sb.Clear().Append('<#Invalid reference: #>').Append(_varInfo.Symbol).ToString()).Pin();
        ELSE
            _progress := _progress + 1;
        END_IF
    END_IF

    IF _progress = 1 THEN
        inoControl.DrivesOn := TRUE;
        inoControl.DrivesOff := _blink.outQ;

        IF NOT inoStatus.State.DrivesReady THEN
            inoControl.DrivesOff := FALSE;
            _progress := 0;
        END_IF
    END_IF

    _varInfo := __VARINFO(inoStatus.State.DrivesReady);

    THIS^.Messenger.OnCondition(_infoTimer.Q)
        .Warning(_sb.Clear().Append('<# Waiting for signal: #>').Append(_varInfo.Symbol).Append('<# is OFF #>').ToString());

    DoneWhen(NOT inoStatus.State.DrivesReady);
    CallTimers(TRUE);
    THIS^.ThrowWhen(_errorTimer.Q);
END_IF;

IF THIS^.Error AND NOT _errorMessage.Pinned THEN
    THIS^.Restore();
END_IF

METHOD PUBLIC FB_init : BOOL
VAR_INPUT
    bInitRetains : BOOL; // if TRUE, the retain variables are initialized (warm start / cold start)
    bInCopyCode : BOOL; // if TRUE, the instance afterwards gets moved into the copy code (online change)
    ParentObject : ITcoObject;
END_VAR
END_METHOD

(*~
    <docu>
        <summary>
            Executes when task is aborted.
        </summary>
    </docu>
~*)
METHOD PROTECTED OnAbort
IF __ISVALIDREF(inoStatus) THEN
    THIS^.inoStatus.ActionDescription := '<#Start at Main was aborted, while not yet completed!#>';
END_IF;
END_METHOD

(*~
    <docu>
        <summary>
            Executes when task reaches the ```Done``` state .
        </summary>
    </docu>
~*)
METHOD PROTECTED OnDone
IF __ISVALIDREF(inoStatus) THEN
    THIS^.inoStatus.ActionDescription := '<#Stop motors was completed successfully.#>';
END_IF;
END_METHOD

(*~
    <docu>
        <summary>
            Executes when task reaches the ```Error``` state.
                </summary>
    </docu>
~*)
METHOD PROTECTED OnError
VAR
    description : STRING;
END_VAR
THIS^.inoStatus.ActionDescription := '<#Stop motors finished with error.#>';

IF __ISVALIDREF(inoStatus) THEN
    THIS^.inoStatus.ActionDescription := description;
END_IF;

THIS^._errorMessage.Error(_sb.Clear().Append(description).Append(' To restore acknowledge this alarm.').ToString()).Pin();
END_METHOD

METHOD PROTECTED OnStart
IF __ISVALIDREF(inoStatus) THEN
    THIS^.inoStatus.ActionDescription := '<#Stop motors started.#>';
END_IF;
END_METHOD

(*~
    <docu>
        <summary>
            Restores this instance to the Ready state. Can be called explicitly or from within one of the restore mechanisms.
            <para>
                See also <see cref="PlcDocu.TcoCore.TcoTask.AutoRestorable()"/>
            </para>
        </summary>
    </docu>
~*)
METHOD Restore : ITcoRestorable
SUPER^.Restore();
END_METHOD

END_FUNCTION_BLOCK
